//Shuttle car element configurations
TYPE ST_CFG_ProBoxElementShuttle EXTENDS ST_CFG_ProBoxElementBase :
(**************************************************************************************
 * 	Application		:	BoxControl Framework
 *	Revision		:	$Revision:  $
 *	Revision date	:	$Date: $
 *	Last changed by	:	$Author: $
 *	URL				:	$URL: $
 *
 *	Purpose			:	Shuttle car element configuration.
 *
 * ------------------------------------------------------------------------------------
 *	Copyright Swisslog [IP AG], Switzerland. All rights reserved.
 * 
 * ------------------------------------------------------------------------------------
 *	
 * 	Revision History: 
 *
 * 	VERSION			DATE			INITIALS			DESCRIPTION
 *
 **************************************************************************************)	
STRUCT
	//BrakeTime				: TIME:=T#1S; 			// Time before the brake is applied after running shuttle car conveyor A or B	
	ConvCFG					: ARRAY[1..GVL_MPD.MAXPDs] OF ST_CFG_PDs_Shuttle; //Configuration settings for Pickup and or Deposit functions to the shuttle car
	TimeOutMove				: TIME := T#30S;		// Shuttle car timeout value
	CvCC					: DINT := 1000;  		// Encoder value, Center to Center distance if shuttle car has 2 conveyors
	EncoderHysterisis		: DINT := 5;			// Encoder fluktuation allowed. default is +- 5mm
	DriveCFG				: ST_CFG_MPD_Drive;	// Shuttle car drive configuration parameters
	EnableIdlePosition		: BOOL;					// Enable Idle position for the shuttle car
	ApEntryPositions		: ARRAY[1..GVL_PB_SG.NUMBER_OF_AP_PANELS] OF DINT; // Entry position [mm] for each AP cabinet
	AkEntryPosition			: DINT; // Entry position [mm] for the AK cabinet
	IdlePosition			: DINT := 500;			// Idle position [mm]			
	TiltLiftTime 			: TIME;
	TiltEnable				: ARRAY[GVL_MPD.CV_A..GVL_MPD.CV_B] OF BOOL;	//Enable Shuttle Car Tilt functionality
 	SgGroupRef				: REFERENCE TO FB_ProBOXSG;
END_STRUCT
END_TYPE

(* stored: Version 1.1.0.1, ProductVersion 3.1.4024.9
   DUT ST_CFG_ProBoxElementShuttle: Id {3ea55ded-b40a-47e4-9438-9f821659e21f} *)
